{attribute addProperty BoxType "AX8206-0000-0041-0041"}
{attribute addProperty Id "Ch_B_Target_torque_forceAT %Q*INT162"}
{attribute addProperty CRC "58827535"}
{attribute addProperty SizeInBites "16"}
{attribute addProperty SizeInBytes "2"}
TYPE Ch_B_TorqueControl_Outputs_0381A30F :
STRUCT
	{attribute addProperty Name "Ch_B_Target_torque_force"}
	Ch_B_Target_torque_force AT %Q* : INT;
END_STRUCT
END_TYPE

(* stored: Version 1.2.0.0, ProductVersion 3.1.4024.9
   DUT Ch_B_TorqueControl_Outputs_0381A30F: Id {f083e577-55f3-4a60-a49c-af7fa2117253} *)
